# EPICS substitutions: blenApp/Db/blenLCLS2.substitutions
########################################################################################################################
# Summary:             Carrier substitutions file to generate PVs for CPSW registers
# Author:              C. Ford <caf@slac.stanford.edu>
# Date:                21-mar-2017
# YAML config version: AmcCarrierBcm_00000018
# Modified:
#                      R. Reno <rreno@slac.stanford.edu>
#                      20-Apr-2020
########################################################################################################################

########################################################################################################################
# Macros:
#   P,R: The PV name as $(P):$(R)
#   DESC, PINI, SCAN, NELM, etc.: The same fields on the records
#   PORT: The asyn port name. It must match the port name given when calling "YCPSWASYNConfig" on st.cmd
#   PARAM: The asyn paramter name. It must be defined in the dictionary file and assigned to a register
########################################################################################################################

#======================================
# Registers with ScalVal_RO interfaces
#======================================
# Single register
file "RegisterIn.template" { pattern
{ P,          R,              DESC,                           PINI,   SCAN,       PORT, EGU,  PARAM            }
{ $(P), DeviceDna,      "Xilinx Device DNA",                      "YES",  "Passive",  $(PORT),   "",   STAT:DeviceDna    }
{ $(P), FpgaVersion,    "FPGA Firmware Version Number",           "YES",  "Passive",  $(PORT),   "",   STAT:FpgaVersion  }
{ $(P), UpTimeCnt,      "Seconds since last reset",               "YES",  "1 second", $(PORT),   "s",  STAT:UpTimeCnt    }
{ $(P), DeviceId,       "Device Identification",                  "YES",  "Passive",  $(PORT),   "",   STAT:DeviceId     }
# BSA status
{ $(P), SofCount,       "BSA: Start of Frame Count",              "YES",  "1 second", $(PORT),   "",   BSA:sofCount      }
{ $(P), EofCount,       "BSA: End of Frame Count",                "YES",  "1 second", $(PORT),   "",   BSA:eofCount      }
{ $(P), CrcErrCount,    "BSA: CRC error count",                   "YES",  "1 second", $(PORT),   "",   BSA:CrcErrCount   }
{ $(P), RxClkCount,     "BSA: Recovered clk count /16",           "YES",  "1 second", $(PORT),   "",   BSA:RxClkCount    }
{ $(P), RxRstCount,     "BSA: Recieve link reset count",          "YES",  "1 second", $(PORT),   "",   BSA:RxRstCount    }
{ $(P), RxDecErrCount,  "BSA: Recieve 8b/10b decode error count", "YES",  "1 second", $(PORT),   "",   BSA:RxDecErrCount }
{ $(P), RxDspErrCount,  "BSA: Recieve disparity error count",     "YES",  "1 second", $(PORT),   "",   BSA:RxDspErrCount }
{ $(P), RxLinkUp,       "BSA: Recieve link status",               "YES",  "1 second", $(PORT),   "",   BSA:RxLinkUp      }
# CmnConfig status
{ $(P), TmitTimeUp,     "TMIT Time Stamp Upper Part",             "YES",  "1 second", $(PORT),   "",   STAT:TmitTimeUp   }
{ $(P), TmitTimeLow,    "TMIT Time Stamp Lower Part",             "YES",  "1 second", $(PORT),   "",   STAT:TmitTimeLow  }
{ $(P), TmitStatus0,    "BPM0 Tmit Status",                       "YES",  "1 second", $(PORT),   "",   STAT:TmitStatus0  }
{ $(P), TmitStatus1,    "BPM1 Tmit Status",                       "YES",  "1 second", $(PORT),   "",   STAT:TmitStatus1  }
{ $(P), TmitTmit0,      "BPM0 Tmit",                              "YES",  "1 second", $(PORT),   "",   STAT:TmitTmit0    }
{ $(P), TmitTmit1,      "BPM1 Tmit",                              "YES",  "1 second", $(PORT),   "",   STAT:TmitTmit1    }
{ $(P), LclTimeUp,      "Local Time Stamp Upper Part",            "YES",  "1 second", $(PORT),   "",   STAT:LclTimeUp    }
{ $(P), LclTimeLow,     "Local Time Stamp Lower Part",            "YES",  "1 second", $(PORT),   "",   STAT:LclTimeLow   }
{ $(P), TmitInvalid,    "",                                       "YES",  "1 second", $(PORT),   "",   STAT:TmitInvalid  }
{ $(P), TmitSmall,      "Indicate TMIT is too small",             "YES",  "1 second", $(PORT),   "",   STAT:TmitSmall    }
{ $(P), StatusOfBsa0,   "",                                       "YES",  "1 second", $(PORT),   "",   STAT:Bsa0         }
{ $(P), StatusOfBsa1,   "",                                       "YES",  "1 second", $(PORT),   "",   STAT:Bsa1         }
{ $(P), StatusOfBsa2,   "",                                       "YES",  "1 second", $(PORT),   "",   STAT:Bsa2         }
# MoverCntl status
{ $(P), StatusLimitSw,  "",                                       "YES",  "1 second", $(PORT),   "",   MVR:StatusLimitSw }
{ $(P), Inserted,       "",                                       "YES",  "1 second", $(PORT),   "",   MVR:Inserted      }
{ $(P), Removed,        "",                                       "YES",  "1 second", $(PORT),   "",   MVR:Removed       }
}

# Array of register
file "RegisterArrayIn.template" { pattern
{ P,          R,             DESC,                          NELM,   PINI,   SCAN,       PORT,  PARAM       }
}

# Array of 8-bit register as a string
file "RegisterArrayChar.template" { pattern
{ P,        R,              DESC,                           NELM,   PINI,   SCAN,       PORT,  PARAM       }
# Shared
{ $(P), BuildStamp,     "Firmware Build String",        256,     "YES",  "Passive",  $(PORT),  STAT:BuildStamp }
}

# ENUM register
file "RegisterEnumBIn.template" { pattern
{ P,        R,              DESC,                    PINI,   ZNAM,       ONAM,       SCAN,      PORT, PARAM     }
}

#======================================
# Register with ScalVal interfaces
#======================================

file "RegisterOut.template" { pattern
{ P,        R,              DESC,                                       PINI,   SCAN,       PORT,  PARAM       }
{ $(P), ScratchPad,     "Register to test R/W"                    "NO",   "Passive",  $(PORT),    :ScratchPad }
# BSA
{ $(P), ClkSel,         "Select between LCLS-I/II timing",        "YES",  "1 second", $(PORT),     TIME:ClkSel }
{ $(P), RxPolarity,     "",                                        "NO",   "Passive",  $(PORT),    BSA:RxPolarity }
{ $(P), PhaseTarget,    "",                                        "NO",   "Passive",  $(PORT),    BSA:PhaseTarget }
# CmnConfig
{ $(P), AppType,        "",                                        "NO",   "Passive",  $(PORT),    CONF:AppType }
{ $(P), CalibEnable,    "",                                        "NO",   "Passive",  $(PORT),    CONF:CalibEnable }
{ $(P), Location,       "",                                        "NO",   "Passive",  $(PORT),    CONF:Location }
{ $(P), SelBpm,         "BPM0/BPM1 Incoming Stream",               "YES",  "1 second", $(PORT),    CONF:SelBpm }
{ $(P), TreshTmit,      "",                                        "NO",   "Passive",  $(PORT),    CONF:TreshTmit }
# MoverCntl
{ $(P), MoverOnOff,     "",                                        "NO",   "Passive",  $(PORT),   MVR:MoverOnOff }
{ $(P), IgnoreMover,    "",                                        "NO",   "Passive",  $(PORT),   MVR:IgnoreMover }
}

file "RegisterOutRBV.template" { pattern
{ P,           R,                DESC,                PINI,      SCAN,      PORT,        PARAM       }
# Shared
{ $(P), ScratchPadRBV,     "Register to test R/W",    "YES",  "1 second",  $(PORT),    :ScratchPad }
# BSA
{ $(P), ClkSelRBV,  "",                                "YES",  "1 second",  $(PORT),    TIME:ClkSel }
{ $(P), RxPolarityRBV,  "",                            "YES",  "1 second",  $(PORT),    BSA:RxPolarity }
{ $(P), PhaseTargetRBV, "",                            "YES",  "1 second",  $(PORT),    BSA:PhaseTarget }
# CmnConfig
{ $(P), AppTypeRBV,     "",                            "YES",  "1 second",  $(PORT),    CONF:AppType }
{ $(P), CalibEnableRBV, "",                            "YES",  "1 second",  $(PORT),    CONF:CalibEnable }
{ $(P), LocationRBV,    "",                            "YES",  "1 second",  $(PORT),    CONF:Location }
{ $(P), SelBpmRBV,      "BPM0/BPM1 Incoming Stream",   "YES",  "1 second",  $(PORT),    CONF:SelBpm }
{ $(P), TreshTmitRBV,   "",                            "YES",  "1 second",  $(PORT),    CONF:TreshTmit }
# MoverCntl
{ $(P), MoverOnOffRBV,  "",                            "YES",  "1 second",  $(PORT),    MVR:MoverOnOff }
{ $(P), IgnoreMoverRBV, "",                            "YES",  "1 second",  $(PORT),    MVR:IgnoreMover }
}

# ENUM register
file "RegisterEnumBOut.template" { pattern
{ P,        R,              DESC,        PINI   ZNAM,        ONAM,     SCAN,       PORT, PARAM     }
}

file "RegisterEnumBOutRBV.template" { pattern
{ P,        R,              DESC,         PINI    ZNAM,        ONAM,     SCAN,        PORT, PARAM     }
}

#======================================
# Register with DoubleVal_RO interfaces
#======================================

file "RegisterDoubleIn.template" { pattern
{ P,              R,            DESC,                         PINI,   SCAN,        PORT,   EGU,    PARAM    }
}

#======================================
# Register with DoubleVal interfaces
#======================================

file "RegisterDoubleOut.template" { pattern
{ P,              R,         DESC,                            PINI,  SCAN,        PORT,     EGU,      PARAM       }
{ $(P), MoverAttenuation,    "",                              "NO",   "Passive",  $(PORT),   "",  MVR:Attenuation }
}

file "RegisterDoubleOutRBV.template" { pattern
{ P,              R,           DESC,                            PINI,  SCAN,        PORT,      EGU,      PARAM       }
{ $(P), MoverAttenuationRBV,    "",                              "NO",   "Passive",  $(PORT),   "",  MVR:Attenuation }
}

#======================================
# Register with Command interfaces
#======================================
file "RegisterCommand.template" { pattern
{ P,            R,            DESC,                            PINI,   SCAN,       PORT,   PARAM   }
}

#======================================
# Register with Stream interfaces
#======================================

file "RegisterStream.template" {pattern
{ P,            R,          DESC,               NELM,       PINI,   PORT,   PARAM       }
}

# For Stream interfaces, an additional parameter is automatically created
# and the name is generated adding ":16" to the original parameter name
# This gives access to the same stream data, but as 16-bit words which
# is the case for ADC samples for example. Note that the NELM is 2x

file "RegisterStream16.template" {pattern
{ P,            R,          DESC,                           NELM,        PINI,  PORT,  PARAM         }
}
